// TIA Portal V16 export
// export: Created 2021-11-12T13:31:53.6986853Z, ExportSetting WithDefaults, DisplayName Totally Integrated Automation Portal, DisplayVersion V16 Update 3, DisplayName TIA Portal Version Control Interface, DisplayVersion V16 Update 2, DisplayName TIA Portal Openness, DisplayVersion V16 Update 3, DisplayName SINAMICS Startdrive Advanced, DisplayVersion V16 Update 5, DisplayName SINAMICS Startdrive G130, G150, S120, S150, SINAMICS MV, S210, DisplayVersion V16 Update 5, DisplayName SINAMICS Startdrive G110M, G120, G120C, G120D, G120P, G115D, DisplayVersion V16 Update 5, DisplayName STEP 7 Professional, DisplayVersion V16 Update 3, DisplayName STEP 7 Safety, DisplayVersion V16, DisplayName WinCC UA Professional, DisplayVersion V16 Update 3
FUNCTION_BLOCK "StationMEM1"   // FB73, LAD
{ S7_Optimized_Access := 'TRUE' }
VERSION : 0.1
// stored: AutoNumber true, IsIECCheckEnabled false, IsRetainMemResEnabled false, MemoryReserve 100, SetENOAutomatically false, UDAEnableTagReadback false
   VAR_INPUT
      IS_Inputs : "UDT_COMM_MEM1_CRS";   // Input structure from blasting machine THM1
   END_VAR
   VAR_OUTPUT
      OS_Outputs : "UDT_COMM_CRS_MEM1";   // Output structure for blasting machine THM1
   END_VAR
   VAR
      SF_Alarm1 : "STD_DI_Mon";
      SF_Alarm2 : "STD_DI_Mon";
      SF_Alarm3 : "STD_DI_Mon";
      SF_Alarm4 : "STD_DI_Mon";
      SF_Alarm5 : "STD_DI_Mon";
      SF_Alarm6 : "STD_DI_Mon";
      SF_Alarm7 : "STD_DI_Mon";
      SF_Alarm8 : "STD_DI_Mon";
      SS_Edge : Array[0..15] of Bool;   // Edge evalution
   END_VAR
   VAR_TEMP
      TB1PwrOk : Bool;   // Station powered
      TB1SetParam : Bool;   // Set loaded parameters memory
   END_VAR
   VAR_TEMP   // added for the SCL form of the ladder/FBD networks
      _w1 : Bool;
      _w2 : Bool;
   END_VAR
BEGIN

REGION Network 1: *************** Alarms ***************
END_REGION

REGION Network 2: Power OK
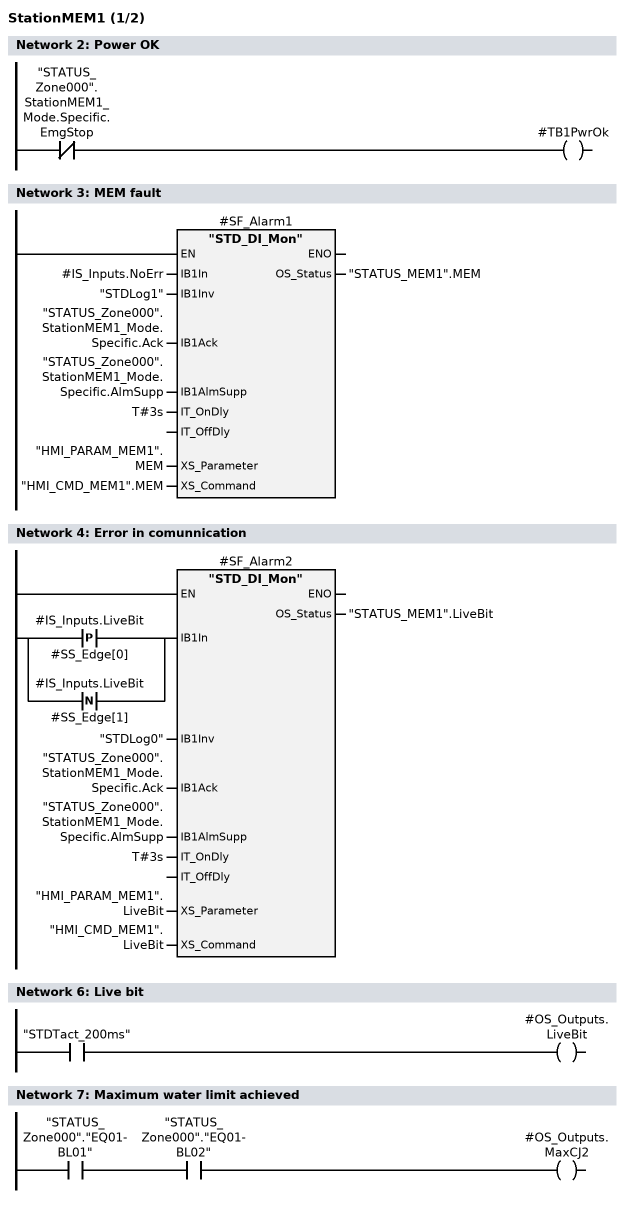
   RUNG wire#powerrail
      I_Contact( "STATUS_Zone000".StationMEM1_Mode.Specific.EmgStop )
      Coil( #TB1PwrOk )
   END_RUNG
   // the same network as SCL:
   #TB1PwrOk := NOT "STATUS_Zone000".StationMEM1_Mode.Specific.EmgStop;
END_REGION

REGION Network 3: MEM fault
   RUNG wire#powerrail
      #SF_Alarm1(IB1In := #IS_Inputs.NoErr, IB1Inv := "STDLog1", IB1Ack := "STATUS_Zone000".StationMEM1_Mode.Specific.Ack, IB1AlmSupp := "STATUS_Zone000".StationMEM1_Mode.Specific.AlmSupp, IT_OnDly := T#3s, IT_OffDly :=, XS_Parameter := "HMI_PARAM_MEM1".MEM, XS_Command := "HMI_CMD_MEM1".MEM, OS_Status => "STATUS_MEM1".MEM)
   END_RUNG
   // the same network as SCL:
   #SF_Alarm1(IB1In := #IS_Inputs.NoErr,   // "STD_DI_Mon"
              IB1Inv := "STDLog1",
              IB1Ack := "STATUS_Zone000".StationMEM1_Mode.Specific.Ack,
              IB1AlmSupp := "STATUS_Zone000".StationMEM1_Mode.Specific.AlmSupp,
              IT_OnDly := T#3s,
              XS_Parameter := "HMI_PARAM_MEM1".MEM,
              XS_Command := "HMI_CMD_MEM1".MEM,
              OS_Status => "STATUS_MEM1".MEM);
END_REGION

REGION Network 4: Error in comunnication
   RUNG wire#powerrail
      #SF_Alarm2(IB1In := wire#w1, IB1Inv := "STDLog0", IB1Ack := "STATUS_Zone000".StationMEM1_Mode.Specific.Ack, IB1AlmSupp := "STATUS_Zone000".StationMEM1_Mode.Specific.AlmSupp, IT_OnDly := T#3s, IT_OffDly :=, XS_Parameter := "HMI_PARAM_MEM1".LiveBit, XS_Command := "HMI_CMD_MEM1".LiveBit, OS_Status => "STATUS_MEM1".LiveBit)
   END_RUNG
   RUNG wire#powerrail
      P_Contact(operand := #IS_Inputs.LiveBit, bit := #SS_Edge[0])
   END_RUNG wire#w1
   RUNG wire#powerrail
      N_Contact(operand := #IS_Inputs.LiveBit, bit := #SS_Edge[1])
   END_RUNG wire#w1
   // the same network as SCL:
   #_w1 := #IS_Inputs.LiveBit AND NOT #SS_Edge[0];   // rising edge of #IS_Inputs.LiveBit
   #SS_Edge[0] := #IS_Inputs.LiveBit;
   #_w2 := NOT #IS_Inputs.LiveBit AND #SS_Edge[1];   // falling edge of #IS_Inputs.LiveBit
   #SS_Edge[1] := #IS_Inputs.LiveBit;
   #SF_Alarm2(IB1In := #_w1 OR #_w2,   // "STD_DI_Mon"
              IB1Inv := "STDLog0",
              IB1Ack := "STATUS_Zone000".StationMEM1_Mode.Specific.Ack,
              IB1AlmSupp := "STATUS_Zone000".StationMEM1_Mode.Specific.AlmSupp,
              IT_OnDly := T#3s,
              XS_Parameter := "HMI_PARAM_MEM1".LiveBit,
              XS_Command := "HMI_CMD_MEM1".LiveBit,
              OS_Status => "STATUS_MEM1".LiveBit);
END_REGION

REGION Network 5: *************** Interface to water managment system ***************
END_REGION

REGION Network 6: Live bit
   RUNG wire#powerrail
      Contact( "STDTact_200ms" )
      Coil( #OS_Outputs.LiveBit )
   END_RUNG
   // the same network as SCL:
   #OS_Outputs.LiveBit := "STDTact_200ms";
END_REGION

REGION Network 7: Maximum water limit achieved
   RUNG wire#powerrail
      Contact( "STATUS_Zone000"."EQ01-BL01" )
      Contact( "STATUS_Zone000"."EQ01-BL02" )
      Coil( #OS_Outputs.MaxCJ2 )
   END_RUNG
   // the same network as SCL:
   #OS_Outputs.MaxCJ2 := "STATUS_Zone000"."EQ01-BL01" AND "STATUS_Zone000"."EQ01-BL02";
END_REGION

REGION Network 8: Some part of line in production mode
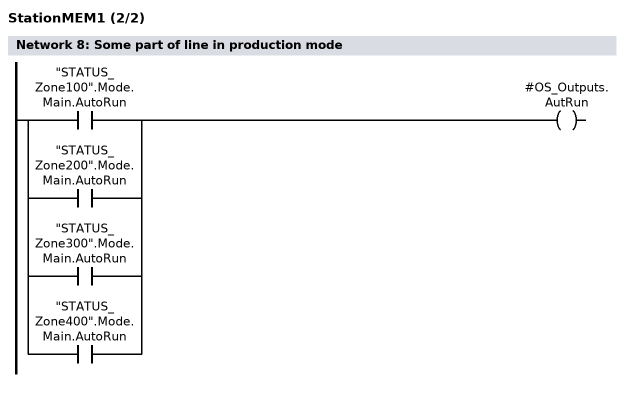
   RUNG wire#powerrail
      Contact( "STATUS_Zone100".Mode.Main.AutoRun )
      wire#w1
      Coil( #OS_Outputs.AutRun )
   END_RUNG
   RUNG wire#powerrail
      Contact( "STATUS_Zone200".Mode.Main.AutoRun )
   END_RUNG wire#w1
   RUNG wire#powerrail
      Contact( "STATUS_Zone300".Mode.Main.AutoRun )
   END_RUNG wire#w1
   RUNG wire#powerrail
      Contact( "STATUS_Zone400".Mode.Main.AutoRun )
   END_RUNG wire#w1
   // the same network as SCL:
   #OS_Outputs.AutRun := "STATUS_Zone100".Mode.Main.AutoRun OR "STATUS_Zone200".Mode.Main.AutoRun OR "STATUS_Zone300".Mode.Main.AutoRun OR "STATUS_Zone400".Mode.Main.AutoRun;
END_REGION
END_FUNCTION_BLOCK
